// TIA Portal project "Task_5" (V18)

(* hardware
DEVICE "S7-1500/ET200MP station_1"  S7-1500 station
   slot 0: "导轨_0"  Rack  6ES7 590-1***0-0AA0
   slot 1: "PLC_1"  CPU 1516-3 PN/DP  6ES7 516-3AN01-0AB0  V2.6
      slot 3: "CPU 显示_1"  6ES7591-1BA00-0AA0
      slot 32768: "PROFINET 接口_1"  X1
      slot 33024: "PROFINET 接口_2"  X2
      slot 33280: "DP 接口_1"  X3
   slot 2: "DI 32x24VDC HF_1"  DI 32x24VDC HF  6ES7 521-1BL00-0AB0  V2.1
   slot 3: "DQ 32x24VDC/0.5A HF_1"  DQ 32x24VDC/0.5A HF  6ES7 522-1BL01-0AB0  V1.1
   slot 4: "AI 8xU/I/RTD/TC ST_1"  AI 8xU/I/RTD/TC ST  6ES7 531-7KF00-0AB0  V2.2
   slot 5: "AQ 4xU/I ST_1"  AQ 4xU/I ST  6ES7 532-5HD00-0AB0  V2.2
*)

// ===== PLC "PLC_1"  CPU 1516-3 PN/DP =====

VAR_GLOBAL   // PLC tag table "默认变量表"
   "按键总数" AT %MW100 : Word;
   "按钮A" AT %I1.0 : Bool;
   "按钮B" AT %I1.1 : Bool;
   "按钮A次数" AT %MW102 : Word;
   "按钮B次数" AT %MW104 : Word;
   "绿灯" AT %Q1.2 : Bool;
   "红灯" AT %Q1.3 : Bool;
   "黄灯" AT %Q1.1 : Bool;
   "Tag_1" AT %M10.0 : Bool;
   "Tag_2" AT %M10.1 : Bool;
END_VAR

ORGANIZATION_BLOCK "Main"   // OB1, LAD, ProgramCycle
TITLE = "Main Program Sweep (Cycle)"
{ S7_Optimized_Access := 'TRUE' }
VERSION : 0.1
   VAR_INPUT
      Initial_Call : Bool;   // Initial call of this OB
      Remanence : Bool;   // =True, if remanent data are available
   END_VAR
   VAR_TEMP   // added for the SCL form of the ladder/FBD networks
      _w1 : Bool;
      _w2 : Bool;
   END_VAR
BEGIN

REGION Network 1
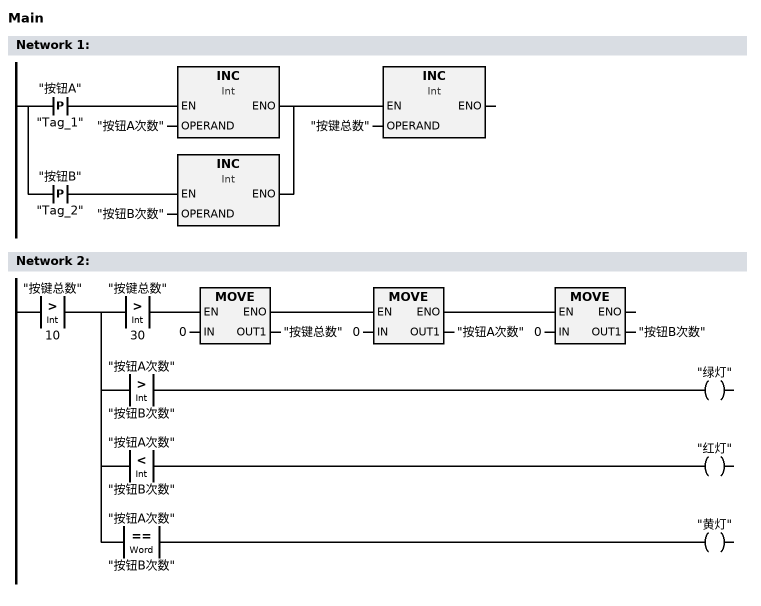
   RUNG wire#powerrail
      P_Contact(operand := "按钮A", bit := "Tag_1")
      { S7_Templates := "DestType := Int" } Inc( "按钮A次数" )
      wire#w1
      { S7_Templates := "DestType := Int" } Inc( "按键总数" )
   END_RUNG
   RUNG wire#powerrail
      P_Contact(operand := "按钮B", bit := "Tag_2")
      { S7_Templates := "DestType := Int" } Inc( "按钮B次数" )
   END_RUNG wire#w1
   // the same network as SCL:
   #_w1 := "按钮A" AND NOT "Tag_1";   // rising edge of "按钮A"
   "Tag_1" := "按钮A";
   IF #_w1 THEN "按钮A次数" := "按钮A次数" + 1; END_IF;
   #_w2 := "按钮B" AND NOT "Tag_2";   // rising edge of "按钮B"
   "Tag_2" := "按钮B";
   IF #_w2 THEN "按钮B次数" := "按钮B次数" + 1; END_IF;
   IF #_w1 OR #_w2 THEN "按键总数" := "按键总数" + 1; END_IF;
END_REGION

REGION Network 2
   RUNG wire#powerrail
      { S7_Templates := "SrcType := Int" } GT_Contact(in1 := "按键总数", in2 := 10)
      wire#w1
      { S7_Templates := "SrcType := Int" } GT_Contact(in1 := "按键总数", in2 := 30)
      Move(in := 0, out1 => "按键总数")
      Move(in := 0, out1 => "按钮A次数")
      Move(in := 0, out1 => "按钮B次数")
   END_RUNG
   RUNG wire#w1
      { S7_Templates := "SrcType := Int" } GT_Contact(in1 := "按钮A次数", in2 := "按钮B次数")
      Coil( "绿灯" )
   END_RUNG
   RUNG wire#w1
      { S7_Templates := "SrcType := Int" } LT_Contact(in1 := "按钮A次数", in2 := "按钮B次数")
      Coil( "红灯" )
   END_RUNG
   RUNG wire#w1
      { S7_Templates := "SrcType := Word" } EQ_Contact(in1 := "按钮A次数", in2 := "按钮B次数")
      Coil( "黄灯" )
   END_RUNG
   // the same network as SCL:
   #_w1 := "按键总数" > 10;
   #_w2 := #_w1 AND ("按键总数" > 30);
   IF #_w2 THEN
       "按键总数" := 0;
       "按钮A次数" := 0;
       "按钮B次数" := 0;
   END_IF;
   "绿灯" := #_w1 AND ("按钮A次数" > "按钮B次数");
   "红灯" := #_w1 AND ("按钮A次数" < "按钮B次数");
   "黄灯" := #_w1 AND ("按钮A次数" = "按钮B次数");
END_REGION
END_ORGANIZATION_BLOCK